{attribute 'qualified_only'}
{attribute 'strict'}
TYPE HighLevelCondition :
(
	INIT,
	RUN,
	SLEEP
);
END_TYPE

(* stored: Version 1.1.0.1, ProductVersion 3.1.4024.12
   DUT HighLevelCondition: Id {dcaebc43-7ee5-463b-bf6d-8ef9d0a436df} *)
